FUNCTION_BLOCK FB_Zentral
VAR_INPUT
END_VAR
VAR_OUTPUT
END_VAR
VAR
END_VAR

END_FUNCTION_BLOCK

(* stored: Version 1.1.0.1, ProductVersion 3.1.4024.9
   POU FB_Zentral: Id {5500bd56-900a-4008-9aef-26bedbb9cf7c}, SpecialFunc None *)
